(* IEC 61131-3 sources: AXOpen/src/templates.simple/ax/src/templates/unit, 9 files *)

(* ---- AutomatSequence.st ---- *)
NAMESPACE axosimple.UnitTemplate
    USING axosimple;
    USING AXOpen.Data;
    USING AXOpen.Core;
    USING System.Strings;

    ///<summary>
    /// Provides automatic mode sequence.
    ///</summary>
    {#ix-set:AttributeName = "<#AUTOMAT#>"}
    {S7.extern=ReadWrite}
    CLASS PUBLIC AutomatSequence
        EXTENDS AXOpen.Core.AxoSequencerContainer
        IMPLEMENTS IModeContainer
        VAR PUBLIC
            Steps : ARRAY[0..150] OF AXOpen.Core.AxoStep;
        END_VAR
        VAR PRIVATE
            Objs : REF_TO axosimple.UnitTemplate.UnitObjects;
            Components : REF_TO axosimple.UnitTemplate.Components;
            ProcessDataManager : REF_TO axosimple.UnitTemplate.ProcessDataManager;
            ProcessSettingsManager : REF_TO axosimple.UnitTemplate.FragmentProcessDataManger;
            TechnologySettingsManager : REF_TO axosimple.UnitTemplate.TechnologyDataManager;

            EntityHeader : REF_TO axosimple.EntityData;
            ProcessData : REF_TO axosimple.UnitTemplate.ProcessData;
            ProcessSettings : REF_TO axosimple.UnitTemplate.ProcessData;
            TechnologySettings : REF_TO axosimple.UnitTemplate.TechnologyData;

            _currentId : STRING;
        END_VAR

        METHOD INTERNAL Run
            VAR_INPUT
                _parent :  AXOpen.Core.IAxoObject;
                _unitObjects : REF_TO axosimple.UnitTemplate.UnitObjects;
            END_VAR

            IF Objs = NULL THEN
                Objs := _unitObjects;

                Components := Objs^.Components;
                ProcessDataManager := Objs^.ProcessData;
                ProcessSettingsManager := Objs^.ProcessSettings;
                TechnologySettingsManager := Objs^.TechnologySettings;

                EntityHeader := REF(ProcessDataManager^.Shared.Entity);
                ProcessData :=  REF(ProcessDataManager^.DataManger.Payload);
                ProcessSettings :=  REF(ProcessSettingsManager^.Payload);
                TechnologySettings :=  REF(TechnologySettingsManager^.DataManger.Payload);

            END_IF;

            SUPER.Run(_parent);
        END_METHOD
        ///<summary>
        /// Contains logic of the steps of this sequence
        ///</summary>

        METHOD OVERRIDE Main
            IF (Components = NULL OR ProcessDataManager = NULL) THEN
                RETURN;
            END_IF;

            // This sequecner executes the steps in cycles from top to bottom
            // in the same order they are written in the program
            // Each step in the sequence must can be used only once.
            // This sets the sequence to run in cycles (top-botton-top and again).
            THIS.SequenceMode := eAxoSequenceMode#Cyclic;

            IF (Steps[0].Execute(THIS, TRUE, '<#GET ID#>')) THEN
                //-------------------------------------------------------
                _currentId := 'newProducedPart';
                THIS.MoveNext();
                //-------------------------------------------------------
            END_IF;

            IF (Steps[10].Execute(THIS, TRUE, '<#GET DATA#>')) THEN
                //-------------------------------------------------------
                // IF(ProcessSettingsManager^.Read('MODEL_S').IsDone()) THEN
                //     ProcessDataManager^.DataManger.Payload := ProcessSettingsManager^.Payload;
                //     THIS.MoveNext();
                // END_IF;

                IF (ProcessDataManager^.CreateOrUpdate(_currentId).IsDone()) THEN
                    THIS.MoveNext();
                END_IF;

                //-------------------------------------------------------
            END_IF;

            IF (Steps[20].Execute(THIS, TRUE, '<#DO SOMETHING#>')) THEN
                //-------------------------------------------------------

                IF(THIS.ProcessDataManager^.DataManger.Payload.JigDataMatrixCode.Inspect(THIS, '').Done()) THEN
                    THIS.MoveNext();
                END_IF;
                //-------------------------------------------------------
            END_IF;

            IF (Steps[30].Execute(THIS, TRUE, '<#DO SOMETHING#>')) THEN
                //-------------------------------------------------------
                IF(THIS.ProcessDataManager^.DataManger.Payload.PartPresence.Inspect(THIS, TRUE).Done()) THEN
                    THIS.MoveNext();
                END_IF;
                //-------------------------------------------------------
            END_IF;

            IF (Steps[4].Execute(THIS, TRUE, '<#DO SOMETHING#>')) THEN
                //-------------------------------------------------------
                IF(THIS.ProcessDataManager^.DataManger.Payload.RivetingPreasure.Inspect(THIS, 1.5).Done()) THEN
                    THIS.MoveNext();
                END_IF;
                //-------------------------------------------------------
            END_IF;

            IF (Steps[149].Execute(THIS, TRUE, '<#UPDATE DATA#>')) THEN
                //-------------------------------------------------------
                IF (ProcessDataManager^.Update(_currentId).IsDone()) THEN
                    THIS.MoveNext();
                END_IF;
                //-------------------------------------------------------
            END_IF;

            // This will close the sequence and will return to the first step.
            THIS.Close(Steps[150]);
        END_METHOD
    END_CLASS
END_NAMESPACE

(* ---- Comonents.st ---- *)
NAMESPACE axosimple.UnitTemplate
    USING axosimple;
    USING AXOpen.Data;
    USING AXOpen.Core;
    USING System.Strings;

    ///<summary>
    /// Groups components of this controller unit.
    ///</summary>
    CLASS Components
        EXTENDS AXOpen.Core.AxoObject
        VAR PUBLIC
            // HERE DECLARE COMPONENTS USED BY THIS CONTROLLED UNIT
            HorizontalCylinder : AXOpen.Components.Pneumatics.AxoCylinder;
            VerticalCylinder : AXOpen.Components.Pneumatics.AxoCylinder;
            GripperCylinder : AXOpen.Components.Pneumatics.AxoCylinder;
            DMCReader : AXOpen.Components.Cognex.Vision.v_6_0_0_0.AxoDataman;
            PartPresenceSensor : AXOpen.Elements.AxoDi;
        END_VAR

        METHOD PUBLIC Update
            VAR_INPUT
                parent : IAxoObject;
            END_VAR
            VAR_IN_OUT
                Inputs : axosimple.Inputs;
                Outputs : axosimple.Outputs;
            END_VAR
            THIS.Initialize(parent);
            // HERE INITIALIZE YOUR COMPONENTS
            HorizontalCylinder.Run(THIS, Inputs.B0[0], Inputs.B0[1], Outputs.B0[0], Outputs.B0[1]);
            VerticalCylinder.Run(THIS, Inputs.B0[2], Inputs.B0[3], Outputs.B0[2], Outputs.B0[3]);
            GripperCylinder.Run(THIS, Inputs.B0[4], Inputs.B0[5], Outputs.B0[4], Outputs.B0[5]);

        END_METHOD
    END_CLASS
END_NAMESPACE

(* ---- Components.st ---- *)
NAMESPACE axosimple.UnitTemplate
    USING axosimple;
    USING AXOpen.Data;
    USING AXOpen.Core;
    USING System.Strings;

    ///<summary>
    /// Groups components of this controller unit.
    ///</summary>
    {S7.extern=ReadWrite}
    CLASS Components
        EXTENDS AXOpen.Core.AxoObject
        VAR PUBLIC
            // HERE DECLARE COMPONENTS USED BY THIS CONTROLLED UNIT
            DI_1 : AXOpen.Elements.AxoDi;
            DI_2 : AXOpen.Elements.AxoDi;
            // DI_3 : AXOpen.Elements.AxoDi;
            // DI_4 : AXOpen.Elements.AxoDi;

            DO_1 : AXOpen.Elements.AxoDo;
            DO_2 : AXOpen.Elements.AxoDo;
            // DO_3 : AXOpen.Elements.AxoDo;
            // DO_4 : AXOpen.Elements.AxoDo;

            AI_1 : AXOpen.Elements.AxoAi;
            AI_2 : AXOpen.Elements.AxoAi;
            // AI_3 : AXOpen.Elements.AxoAi;
            // AI_4 : AXOpen.Elements.AxoAi;

            AO_1 : AXOpen.Elements.AxoAo;
            AO_2 : AXOpen.Elements.AxoAo;
            // AO_3 : AXOpen.Elements.AxoAo;
            // AO_4 : AXOpen.Elements.AxoAo;

            Cylinder_1 : AXOpen.Components.Pneumatics.AxoCylinder;
            Cylinder_2 : AXOpen.Components.Pneumatics.AxoCylinder;
            // Cylinder_3 : AXOpen.Components.Pneumatics.AxoCylinder;
            // Cylinder_4 : AXOpen.Components.Pneumatics.AxoCylinder;

            Reader_1 : AXOpen.Components.Cognex.Vision.v_6_0_0_0.AxoDataman;
            Reader_2 : AXOpen.Components.Cognex.Vision.v_6_0_0_0.AxoDataman;

            Camera_1 : AXOpen.Components.Cognex.Vision.v_6_0_0_0.AxoInsight;
            Camera_2 : AXOpen.Components.Cognex.Vision.v_6_0_0_0.AxoInsight;

            {#ix-attr:[Container(Layout.Stack)]}
            Drive_R1  : AXOpen.Components.Rexroth.Drives.AxoIndraDrive;

            {#ix-attr:[Container(Layout.Stack)]}
            Drive_R2  : AXOpen.Components.Rexroth.Drives.AxoIndraDrive;

            {#ix-attr:[Container(Layout.Stack)]}
            Drive_F1  : AXOpen.Components.Festo.Drives.AxoCmmtAs;

            {#ix-attr:[Container(Layout.Stack)]}
            Drive_F2  : AXOpen.Components.Festo.Drives.AxoCmmtAs;

            _enable         : BOOL := TRUE;
            _enablePositive : BOOL := TRUE;
            _enableNegative : BOOL := TRUE;
        END_VAR

        METHOD PUBLIC Update
            VAR_INPUT
                parent : IAxoObject;
                Inputs : ref_to axosimple.Inputs; // must be a ref_to due to arrays in components
                Outputs : ref_to axosimple.Outputs;
            END_VAR
            THIS.Initialize(parent);

            THIS.Initialize(parent);
            // HERE INITIALIZE YOUR COMPONENTS

            DI_1.Run(THIS, Inputs^.D0[0]);
            DI_2.Run(THIS, Inputs^.D0[0]);
            // DI_3.Run(THIS, Inputs^.D0[0]);
            // DI_4.Run(THIS, Inputs^.D0[0]);

            DO_1.Run(THIS, Outputs^.D0[0]);
            DO_2.Run(THIS, Outputs^.D0[0]);
            // DO_3.Run(THIS, Outputs^.D0[0]);
            // DO_4.Run(THIS, Outputs^.D0[0]);

            AI_1.Run(THIS, Inputs^.A0[0]);
            AI_2.Run(THIS, Inputs^.A0[0]);
            // AI_3.Run(THIS, Inputs^.A0[0]);
            // AI_4.Run(THIS, Inputs^.A0[0]);

            AO_1.Run(THIS, Outputs^.A0[0]);
            AO_2.Run(THIS, Outputs^.A0[0]);
            // AO_3.Run(THIS, Outputs^.A0[0]);
            // AO_4.Run(THIS, Outputs^.A0[0]);

            Cylinder_1.Run(THIS, Inputs^.P0[0], Inputs^.P0[1], Outputs^.P0[0], Outputs^.P0[1]);
            Cylinder_2.Run(THIS, Inputs^.P0[2], Inputs^.P0[3], Outputs^.P0[2], Outputs^.P0[3]);
            // Cylinder_3.Run(THIS, Inputs^.P0[4], Inputs^.P0[5], Outputs^.P0[4], Outputs^.P0[5]);
            // Cylinder_4.Run(THIS, Inputs^.P0[6], Inputs^.P0[7], Outputs^.P0[6], Outputs^.P0[7]);

            Reader_1.Run(parent                     :=  THIS,
            refAcquisitionStatus       :=  REF(Inputs^.Reader_1_Acquisition_Status_1),
            refResultsStatus           :=  REF(Inputs^.Reader_1_Results_Status_1),
            refSoftEventStatus         :=  REF(Inputs^.Reader_1_Soft_Event_Control_1),
            refResultData              :=  REF(Inputs^.Reader_1_Result_Data_128_bytes_1),
            refAcquisitionControl      :=  REF(Outputs^.Reader_1_Acquisition_Control_1),
            refResultsControl          :=  REF(Outputs^.Reader_1_Results_Control_1),
            refSoftEventControl        :=  REF(Outputs^.Reader_1_Soft_Event_Control_1),
            refUserData                :=  REF(Outputs^.Reader_1_User_Data_128_bytes_1));

            Reader_2.Run(parent                     :=  THIS,
            refAcquisitionStatus       :=  REF(Inputs^.Reader_2_Acquisition_Status_1),
            refResultsStatus           :=  REF(Inputs^.Reader_2_Results_Status_1),
            refSoftEventStatus         :=  REF(Inputs^.Reader_2_Soft_Event_Control_1),
            refResultData              :=  REF(Inputs^.Reader_2_Result_Data_128_bytes_1),
            refAcquisitionControl      :=  REF(Outputs^.Reader_2_Acquisition_Control_1),
            refResultsControl          :=  REF(Outputs^.Reader_2_Results_Control_1),
            refSoftEventControl        :=  REF(Outputs^.Reader_2_Soft_Event_Control_1),
            refUserData                :=  REF(Outputs^.Reader_2_User_Data_128_bytes_1));

            Camera_1.Run(parent                  :=  THIS,
            refAcquisitionStatus    :=  REF(Inputs^.Camera_1_Acquisition_Status_1),
            refInspectionStatus     :=  REF(Inputs^.Camera_1_Inspection_Status_1),
            refCommandStatus        :=  REF(Inputs^.Camera_1_Command_Control_1),
            refSoftEventStatus      :=  REF(Inputs^.Camera_1_SoftEvent_Control_1),
            refResultData           :=  REF(Inputs^.Camera_1_Results_64_bytes_1),
            refSoftEventControl     :=  REF(Outputs^.Camera_1_SoftEvent_Control_1),
            refCommandControl       :=  REF(Outputs^.Camera_1_Command_Control_1),
            refInspectionControl    :=  REF(Outputs^.Camera_1_Inspection_Control_1),
            refAcquisitionControl   :=  REF(Outputs^.Camera_1_Acquisition_Control_1),
            refUserData             :=  REF(Outputs^.Camera_1_User_Data_64_bytes_1));

            Camera_2.Run(parent                  :=  THIS,
            refAcquisitionStatus    :=  REF(Inputs^.Camera_2_Acquisition_Status_1),
            refInspectionStatus     :=  REF(Inputs^.Camera_2_Inspection_Status_1),
            refCommandStatus        :=  REF(Inputs^.Camera_2_Command_Control_1),
            refSoftEventStatus      :=  REF(Inputs^.Camera_2_SoftEvent_Control_1),
            refResultData           :=  REF(Inputs^.Camera_2_Results_64_bytes_1),
            refSoftEventControl     :=  REF(Outputs^.Camera_2_SoftEvent_Control_1),
            refCommandControl       :=  REF(Outputs^.Camera_2_Command_Control_1),
            refInspectionControl    :=  REF(Outputs^.Camera_2_Inspection_Control_1),
            refAcquisitionControl   :=  REF(Outputs^.Camera_2_Acquisition_Control_1),
            refUserData             :=  REF(Outputs^.Camera_2_User_Data_64_bytes_1));

            Drive_R1.Run(parent:=THIS,
                refParameter_In     :=  REF(Inputs^.Drive_R1_ParamCh_IDN_1),
                refFieldbus_In      :=  REF(Inputs^.Drive_R1_Input_9_Words_1),
                refParameter_Out    :=  REF(Outputs^.Drive_R1_ParamCh_IDN_1),
                refFieldbus_Out     :=  REF(Outputs^.Drive_R1_Output_13_Words_1),
                Enable              :=  _enable,
                EnablePositive      :=  _enablePositive,
                EnableNegative      :=  _enableNegative);

            Drive_R2.Run(parent:=THIS,
                refParameter_In     :=  REF(Inputs^.Drive_R2_ParamCh_IDN_1),
                refFieldbus_In      :=  REF(Inputs^.Drive_R2_Input_9_Words_1),
                refParameter_Out    :=  REF(Outputs^.Drive_R2_ParamCh_IDN_1),
                refFieldbus_Out     :=  REF(Outputs^.Drive_R2_Output_13_Words_1),
                Enable              :=  _enable,
                EnablePositive      :=  _enablePositive,
                EnableNegative      :=  _enableNegative);

            Drive_F1.Run(parent               :=  THIS,
                    refTelegram111_In   :=  REF(Inputs^.Drive_F1_Siemens_telegram_111_PZD_12_12),
                    refTelegram750_In   :=  REF(Inputs^.Drive_F1_Siemens_telegram_750_PZD_4_1),
                    refTelegram111_Out  :=  REF(Outputs^.Drive_F1_Siemens_telegram_111_PZD_12_12),
                    refTelegram750_Out  :=  REF(Outputs^.Drive_F1_Siemens_telegram_750_PZD_4_1),
                    MAP_HW_ID           :=  Inputs^.Drive_F1_HwId,
                    Enable              :=  _enable,
                    EnablePositive      :=  _enablePositive,
                    EnableNegative      :=  _enableNegative);

            Drive_F2.Run(parent               :=  THIS,
                    refTelegram111_In   :=  REF(Inputs^.Drive_F2_Siemens_telegram_111_PZD_12_12),
                    refTelegram750_In   :=  REF(Inputs^.Drive_F2_Siemens_telegram_750_PZD_4_1),
                    refTelegram111_Out  :=  REF(Outputs^.Drive_F2_Siemens_telegram_111_PZD_12_12),
                    refTelegram750_Out  :=  REF(Outputs^.Drive_F2_Siemens_telegram_750_PZD_4_1),
                    MAP_HW_ID           :=  Inputs^.Drive_F2_HwId,
                    Enable              :=  _enable,
                    EnablePositive      :=  _enablePositive,
                    EnableNegative      :=  _enableNegative);

        END_METHOD
    END_CLASS
END_NAMESPACE

(* ---- GroundSequence.st ---- *)
NAMESPACE axosimple.UnitTemplate
    USING axosimple;
    USING AXOpen.Data;
    USING AXOpen.Core;
    USING System.Strings;

    ///<summary>
    /// Provides ground mode sequence.
    ///</summary>
    {#ix-set:AttributeName = "<#GROUND#>"}
    CLASS PUBLIC GroundSequence
        EXTENDS AXOpen.Core.AxoSequencerContainer
        VAR PUBLIC
            Steps : ARRAY[0..20] OF AxoStep;
            MoveToWork : AxoTask;
        END_VAR
        VAR PRIVATE
            Components : REF_TO Components;
            ProcessData : REF_TO ProcessDataManager;
            TechnologySettings : REF_TO TechnologyDataManager;
            _currentId : STRING;
        END_VAR

        METHOD INTERNAL Run
            VAR_INPUT
                _components : REF_TO Components;
                _processData : REF_TO ProcessDataManager;
                _technologySettings : REF_TO TechnologyDataManager;
                _parent : IAxoObject;
            END_VAR
            Components := _components;
            ProcessData := _processData;
            TechnologySettings := _technologySettings;
            SUPER.Run(_parent);

            // MoveToWork.Initialize(THIS);

        END_METHOD
        ///<summary>
        /// Contains logic of the steps of this sequence
        ///</summary>

        METHOD PROTECTED OVERRIDE Main
            // IF (Components = NULL OR ProcessData = NULL) THEN
            //     RETURN;
            // END_IF;
            // This sequecner executes the steps in cycles from top to bottom
            // in the same order they are written in the program
            // Each step in the sequence must can be used only once.
            // This sets the sequence to run once (top-botton) and stops with done after closing.
            THIS.SequenceMode := eAxoSequenceMode#RunOnce;

            IF (Steps[0].Execute(THIS, TRUE, '<#RESTORE#>')) THEN
                //-------------------------------------------------------
                    ProcessData^.Restore();
                    THIS.MoveNext();

                    ProcessData^.Shared.Entity.WasReset := true;
                    _currentId := 'lastPartId'; // just for simulation
                //-------------------------------------------------------
            END_IF;

            IF (Steps[1].Execute(THIS, TRUE, '<#READ TECHNOLOGY SETTINS#>')) THEN
                //-------------------------------------------------------
                IF(TechnologySettings^.Read('default').IsDone()) THEN
                    THIS.MoveNext();
                END_IF;
                //-------------------------------------------------------
            END_IF;

            IF (Steps[3].Execute(THIS, TRUE, '<#DO SOMETHING#>')) THEN
                //-------------------------------------------------------
                IF CurrentStep.Duration > TIME#2s THEN
                    THIS.MoveNext();
                END_IF;
                //-------------------------------------------------------
            END_IF;

            IF (Steps[19].Execute(THIS, TRUE, '<#SAVE DATA#>')) THEN
                //-------------------------------------------------------
                    IF(ProcessData^.Update(_currentId).IsDone()) THEN
                        THIS.MoveNext();
                    END_IF;
                //-------------------------------------------------------
            END_IF;

            // This will close the sequence and will return to the first step.
            THIS.Close(Steps[20]);
        END_METHOD
    END_CLASS
END_NAMESPACE

(* ---- ProcessData.st ---- *)
NAMESPACE axosimple.UnitTemplate
    USING axosimple;
    USING AXOpen.Data;
    USING AXOpen.Core;
    USING System.Strings;

    CLASS ProcessData
        EXTENDS AXOpen.Data.AxoDataEntity
        VAR PUBLIC
            CounterDelay : ULINT;
        END_VAR
    END_CLASS
END_NAMESPACE

(* ---- ServiceMode.st ---- *)
NAMESPACE axosimple.UnitTemplate
    USING axosimple;
    USING AXOpen.Data;
    USING AXOpen.Core;
    USING System.Strings;

    ///<summary>
    /// Provides logic for service/manual/maintenance mode.
    ///</summary>
    {#ix-set:AttributeName = "<#SERVICE#>"}
    CLASS PUBLIC ServiceMode
        EXTENDS AXOpen.Core.AxoTask
        ///<summary>
        /// Runs service mode logic. This method must be called cyclically.
        ///</summary>

        METHOD PUBLIC Run
            VAR_INPUT
                parent : IAxoObject;
            END_VAR
            VAR_IN_OUT
                components : Components;
            END_VAR
            THIS.Initialize(parent);
            IF THIS.Execute() THEN
                THIS.Handle(components);
            END_IF;
        END_METHOD

        METHOD PRIVATE Handle
            VAR_IN_OUT
                components : Components;
            END_VAR
            ;
            // HERE CALL LOGIC FOR MANUAL/SERICE OPERATIONS
            components.HorizontalCylinder.ActivateManualControl();
            components.VerticalCylinder.ActivateManualControl();
            components.GripperCylinder.ActivateManualControl();
            components.PartPresenceSensor.ActivateManualControl();
        END_METHOD
    END_CLASS
END_NAMESPACE

(* ---- TechnologyData.st ---- *)
NAMESPACE axosimple.UnitTemplate
    USING axosimple;
    USING AXOpen.Data;
    USING AXOpen.Core;
    USING System.Strings;

    CLASS TechnologyData
        EXTENDS AXOpen.Data.AxoDataEntity
        VAR PUBLIC

            Header : axosimple.TechnologyUnitHeader;

            HeatingTemperature   : REAL;

        END_VAR
    END_CLASS
END_NAMESPACE

(* ---- Unit.st ---- *)
NAMESPACE axosimple.UnitTemplate
    USING axosimple;
    USING AXOpen.Data;
    USING AXOpen.Core;
    USING System.Strings;

    ///<summary>
    /// Represents controlled units and high level task coordination.
    ///</summary>
    {S7.extern=ReadWrite}
    CLASS Unit
        EXTENDS axosimple.BaseUnit.UnitBase
        VAR PUBLIC
            ///<summary>
            /// Provide access to unit objets, that are used into sequnces.
            ///</summary>
            UnitObjects  : axosimple.UnitTemplate.UnitObjects;

            ///<summary>
            /// Ground sequence. Contains logic that brings the unit into initial state.
            ///</summary>
            GroundSequence : axosimple.UnitTemplate.GroundSequence;

            ///<summary>
            /// Automatic sequence. Contains logic for automatic operations of this unit.
            ///</summary>
            AutomatSequence : axosimple.UnitTemplate.AutomatSequence;

            ///<summary>
            /// Service mode contains logic for service/manual operations.
            ///</summary>
            ServiceMode : axosimple.UnitTemplate.ServiceMode;
        END_VAR
        ///<summary>
        /// Runs this unit.
        ///</summary>

        METHOD PUBLIC Run
            VAR_INPUT
                parent : IAxoContext;

                ///<summary>
                /// Hardware input structure
                ///</summary>
                Inputs : REF_TO axosimple.Inputs; // MUST BE AS REF_TO DUE TO COMPONENTS THAT HAS REF TO ARRAYS
                ///<summary>
                /// Hardware output structure
                ///</summary>
                Outputs : REF_TO  axosimple.Outputs;
            END_VAR
            THIS.Initialize(parent);
            THIS.Execute(Inputs, Outputs);
        END_METHOD

        METHOD PRIVATE Execute
            VAR_INPUT
                Inputs : REF_TO axosimple.Inputs;
                Outputs : REF_TO  axosimple.Outputs;
            END_VAR

            // Component I/O immange and management handling.
            UnitObjects.Components^.Update(THIS, Inputs, Outputs);
            // Process data manager
            UnitObjects.ProcessData^.Run(THIS);
            // Process settings data manager
            UnitObjects.ProcessSettings^.Run(THIS);
            // Technology data manager
            UnitObjects.TechnologySettings^.Run(THIS);
            // Handles ground sequence
            GroundSequence.Run(THIS, REF(UnitObjects));

            // Restores other states when Ground executes
            IF (GroundSequence.IsBusy()) THEN
                AutomatSequence.Restore();
                ServiceMode.Restore();
            END_IF;

            // Handles automatic sequence (ground must be previously done)
            AutomatSequence.IsDisabled := GroundSequence.Status <> eAxoTaskState#Done;
            AutomatSequence.Run(THIS, REF(UnitObjects));
            // Handles service/manual mode
            ServiceMode.Run(THIS, UnitObjects.Components^);

            IF ServiceMode.IsBusy() THEN
                GroundSequence.Restore();
                AutomatSequence.Restore();
            END_IF;

            // remember last selected technolgy identifier
            if  (UnitObjects.TechnologySettings^.DataManger.Payload.DataEntityId <> '') THEN
                IF UnitObjects.LastTechnologySettings <> UnitObjects.TechnologySettings^.DataManger.Payload.DataEntityId THEN
                    IF UnitObjects.Global^.PersistentData^.InvokeUpdate(THIS, '') THEN
                        UnitObjects.LastTechnologySettings :=  UnitObjects.TechnologySettings^.DataManger.Payload.DataEntityId;
                    END_IF;
                END_IF;
            END_IF;

        END_METHOD
    END_CLASS

END_NAMESPACE

(* ---- UnitObjects.st ---- *)
NAMESPACE axosimple.UnitTemplate

    USING axosimple;
    USING AXOpen.Data;
    USING AXOpen.Core;
    USING System.Strings;

    {S7.extern=ReadWrite}
    CLASS PUBLIC UnitObjects EXTENDS axosimple.BaseUnit.UnitObjects
        VAR PUBLIC
            ///<summary>
            /// Handles and intializes components used by this unit.
            ///</summary>
            Components : REF_TO axosimple.UnitTemplate.Components;

            ///<summary>
            /// Provides access to process data manager of this unit
            ///</summary>
            ProcessSettings : REF_TO axosimple.UnitTemplate.FragmentProcessDataManger;

            ///<summary>
            /// Provides access to process data manager of this unit
            ///</summary>
            ProcessData : REF_TO axosimple.UnitTemplate.ProcessDataManager;

            ///<summary>
            /// Provides access to process data manager of this unit
            ///</summary>
            TechnologySettings : REF_TO axosimple.UnitTemplate.TechnologyDataManager;

            {#ix-attr:[AXOpen.Data.PersistentAttribute("UnitTemplate")]}
            SpecialSettings : STRING[64] ;

        END_VAR
    END_CLASS

END_NAMESPACE
